# EPICS substitutions: iocBoot/ioc13HG100/pid_slow.substitutions
file "$(STD)/db/pid_control.db"
{
pattern
{P,         PID,       INP,    T,                LOPR,  HOPR,  DRVL,  DRVH,  PREC,   KP,  KI,   KD,  SCAN}
{13HG100:,  PID1,     junk,   HG100:Temperature,   0,    85,     0,    85,    3,     0.2,  3.,   0.,  ".1 second"}
}
